// Mitsubishi GX Works2 project: A01_20260228_0   PLC: Q03UDV

TYPE arrange : STRUCT
  層 : ARRAY [1..5] OF STRING[12] := [5('')];
END_STRUCT END_TYPE

TYPE arrange_Bit : STRUCT
  層 : ARRAY [1..5] OF BOOL;
END_STRUCT END_TYPE

TYPE Master_R : STRUCT
  Stacker_Status : WORD;
  Aut_Process : INT;
  Error_Code : INT;
  Task_Status : WORD;
  現在Task_ID : DWORD;
  Task実行総数 : DINT;
  現在位置走行 : INT;
  現在位置リフト : INT;
  現在位置フォーク : INT;
  現在速度走行 : INT;
  現在速度リフト : INT;
  現在速度フォーク : INT;
  現在モード : INT;
  Heartbeat : INT;
  入庫要求1 : INT;
  入庫要求2 : INT;
  出庫要求1 : INT;
  出庫要求2 : INT;
  トルクX軸 : INT;
  トルクY軸 : INT;
  トルクZ軸 : INT;
  異常X軸 : INT;
  異常Y軸 : INT;
  異常Z軸 : INT;
  現在_列 : INT;
  現在_層 : INT;
  Status_Bit : INT;
  Warning_Code : INT;
END_STRUCT END_TYPE

TYPE Master_W : STRUCT
  Task_Type : WORD;
  Task_ID : DWORD;
  起点棚 : INT;
  起点列 : INT;
  起点層 : INT;
  終点棚 : INT;
  終点列 : INT;
  終点層 : INT;
  搬入ST_NO : INT;
  搬出ST_NO : INT;
  System_Heartbeat : INT;
  B01_搬入可 : INT;
  B02_搬入可 : INT;
  B01_搬出可 : INT;
  B02_搬出可 : INT;
  Mode : INT;
  REST_Cont : INT;
  一時停止_Cont : INT;
  Xj軸定位置 : INT;
  Y軸定位置 : INT;
  Z軸定位置 : INT;
  X軸定位列 : INT;
  Y軸定位層 : INT;
  Control_Bit : INT;
  緊急停止 : INT;
  Spare_16 : INT;
  Spare_17 : INT;
  Spare_18 : INT;
  Spare_19 : INT;
END_STRUCT END_TYPE

TYPE Single_Machine : STRUCT
  Query : BOOL;
  成功 : BOOL;
  棚場所 : INT;
  列場所 : INT;
  層場所 : INT;
  搬出PB : BOOL;
  RFID入力 : STRING[12];
  失敗 : BOOL;
  AGV行先 : INT;
  搬出許可条件 : BOOL;
  搬出口 : INT;
  搬出起点Status : INT;
  搬出終点Status : INT;
  搬入ST_パレットStatus : INT;
  搬出ST_パレットStatus : INT;
  搬出起点Status表示 : BOOL;
  終点搬入Status表示 : BOOL;
  搬入ST_Status表示 : BOOL;
  搬出ST_Status表示 : BOOL;
  空き保管場所検索 : BOOL;
  保管条件可 : BOOL;
  搬入PB : BOOL;
  Command_Status : INT;
END_STRUCT END_TYPE

TYPE Wcs_W : STRUCT
  Task_Type : WORD;
  Task_ID : DWORD;
  起点棚 : INT;
  起点列 : INT;
  起点層 : INT;
  終点棚 : INT;
  終点列 : INT;
  終点層 : INT;
  搬入ST_NO : INT;
  搬出ST_NO : INT;
  System_Heartbeat : INT;
  B01_搬入可 : INT;
  B02_搬入可 : INT;
  B01_搬出可 : INT;
  B02_搬出可 : INT;
  異常リセット : INT;
  Spare_7 : INT;
  Spare_8 : INT;
  Spare_9 : INT;
  Spare_10 : INT;
  B01_AGV進入可 : INT;
  B02_AGV進入可 : INT;
  B01_搬入RFID異常 : INT;
  B01_搬出RFID異常 : INT;
  B02_搬入RFID異常 : INT;
  B02_搬出RFID異常 : INT;
  Spare_17 : INT;
  Spare_18 : INT;
  Spare_19 : INT;
END_STRUCT END_TYPE

// global labels: Global1
VAR_GLOBAL
  Stacker_R : Master_R;
  Stacker_W : Master_W;
  Wcs_W : Wcs_W;
  Alone : Wcs_W;
  Mode AT D450 : INT;
  inventory_1 : ARRAY [1..14] OF arrange;
  inventory_2 : ARRAY [1..14] OF arrange;
  搬入RFID_Coding : STRING[12];
  inventory_Bit1 : ARRAY [1..14] OF arrange_Bit;
  inventory_Bit2 : ARRAY [1..14] OF arrange_Bit;
  在庫クリア AT M205 : BOOL;
  Single_Machine : Single_Machine;
  B01CV_OutID : DWORD;
  B02CV_OutID : DWORD;
  Stacker_Done : BOOL;
END_VAR

PROGRAM 01  // PLC 入力
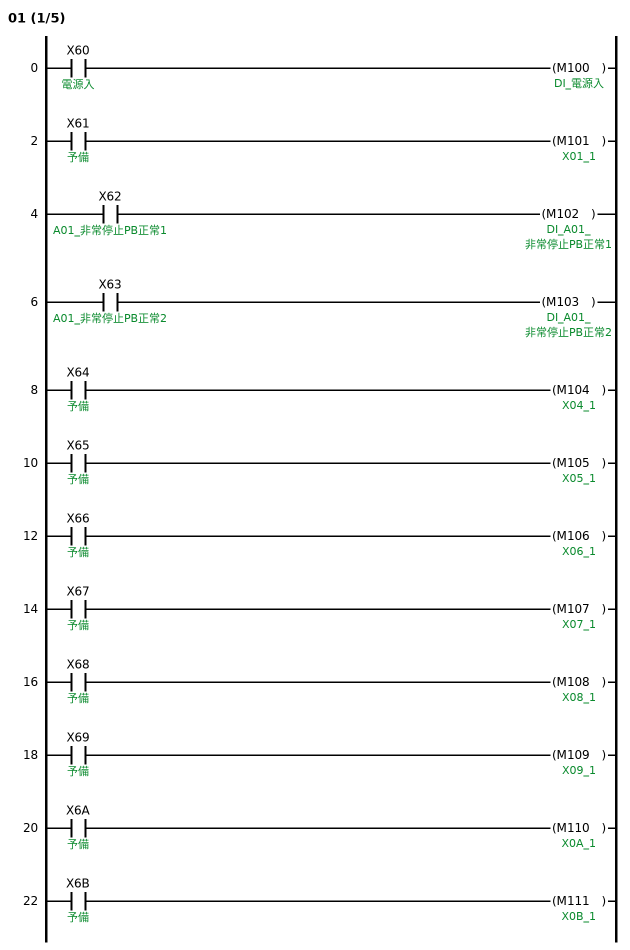
0     LD      X60  ; 電源入
      OUT     M100  ; DI_電源入
2     LD      X61  ; 予備
      OUT     M101  ; X01_1
4     LD      X62  ; A01_非常停止PB正常1
      OUT     M102  ; DI_A01_非常停止PB正常1
6     LD      X63  ; A01_非常停止PB正常2
      OUT     M103  ; DI_A01_非常停止PB正常2
8     LD      X64  ; 予備
      OUT     M104  ; X04_1
10    LD      X65  ; 予備
      OUT     M105  ; X05_1
12    LD      X66  ; 予備
      OUT     M106  ; X06_1
14    LD      X67  ; 予備
      OUT     M107  ; X07_1
16    LD      X68  ; 予備
      OUT     M108  ; X08_1
18    LD      X69  ; 予備
      OUT     M109  ; X09_1
20    LD      X6A  ; 予備
      OUT     M110  ; X0A_1
22    LD      X6B  ; 予備
      OUT     M111  ; X0B_1
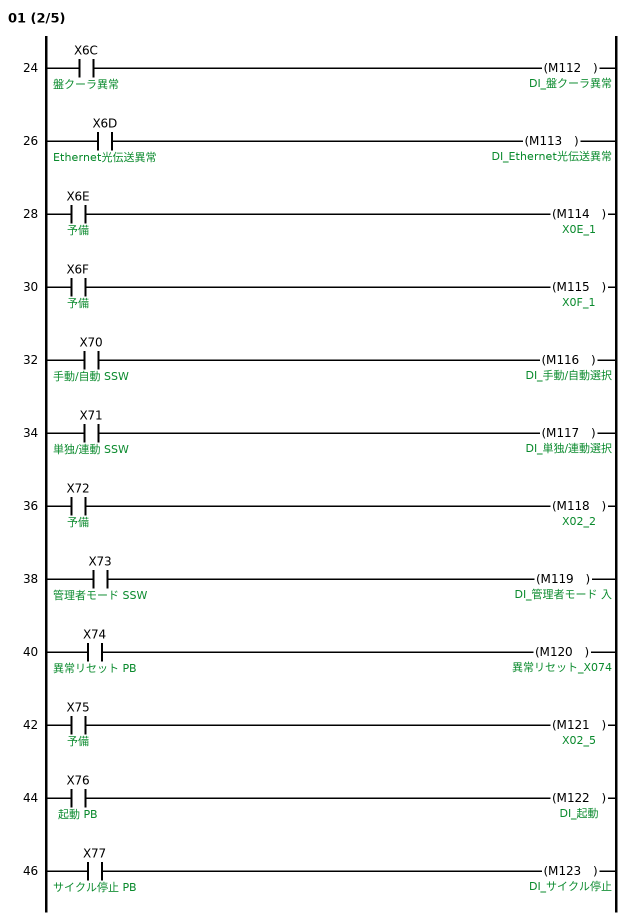
24    LD      X6C  ; 盤クーラ異常
      OUT     M112  ; DI_盤クーラ異常
26    LD      X6D  ; Ethernet光伝送異常
      OUT     M113  ; DI_Ethernet光伝送異常
28    LD      X6E  ; 予備
      OUT     M114  ; X0E_1
30    LD      X6F  ; 予備
      OUT     M115  ; X0F_1
32    LD      X70  ; 手動/自動 SSW
      OUT     M116  ; DI_手動/自動選択
34    LD      X71  ; 単独/連動 SSW
      OUT     M117  ; DI_単独/連動選択
36    LD      X72  ; 予備
      OUT     M118  ; X02_2
38    LD      X73  ; 管理者モード SSW
      OUT     M119  ; DI_管理者モード 入
40    LD      X74  ; 異常リセット PB
      OUT     M120  ; 異常リセット_X074
42    LD      X75  ; 予備
      OUT     M121  ; X02_5
44    LD      X76  ; 起動 PB
      OUT     M122  ; DI_起動
46    LD      X77  ; サイクル停止 PB
      OUT     M123  ; DI_サイクル停止
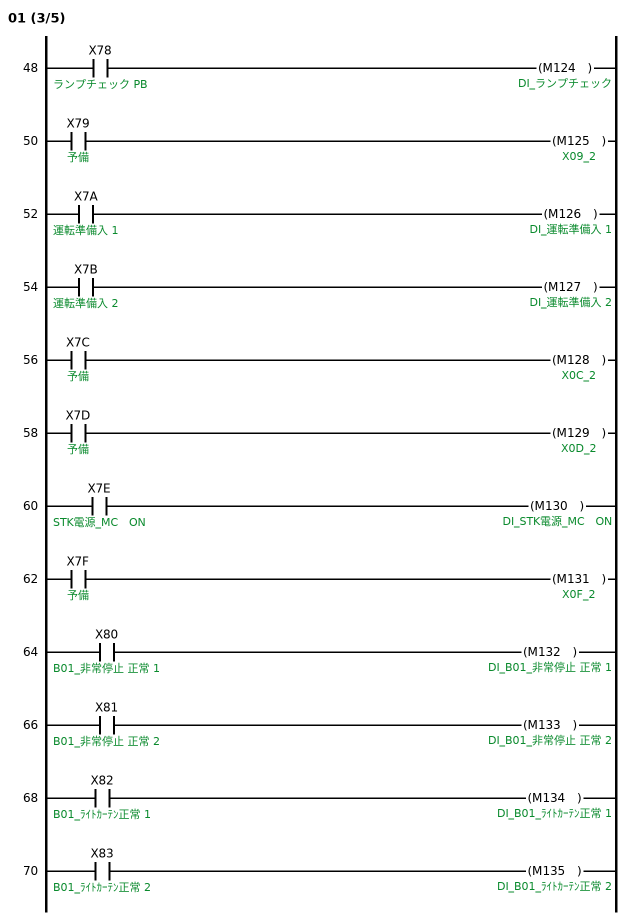
48    LD      X78  ; ランプチェック PB
      OUT     M124  ; DI_ランプチェック
50    LD      X79  ; 予備
      OUT     M125  ; X09_2
52    LD      X7A  ; 運転準備入 1
      OUT     M126  ; DI_運転準備入 1
54    LD      X7B  ; 運転準備入 2
      OUT     M127  ; DI_運転準備入 2
56    LD      X7C  ; 予備
      OUT     M128  ; X0C_2
58    LD      X7D  ; 予備
      OUT     M129  ; X0D_2
60    LD      X7E  ; STK電源_MC　ON
      OUT     M130  ; DI_STK電源_MC　ON
62    LD      X7F  ; 予備
      OUT     M131  ; X0F_2
64    LD      X80  ; B01_非常停止 正常 1
      OUT     M132  ; DI_B01_非常停止 正常 1
66    LD      X81  ; B01_非常停止 正常 2
      OUT     M133  ; DI_B01_非常停止 正常 2
68    LD      X82  ; B01_ﾗｲﾄｶｰﾃﾝ正常 1
      OUT     M134  ; DI_B01_ﾗｲﾄｶｰﾃﾝ正常 1
70    LD      X83  ; B01_ﾗｲﾄｶｰﾃﾝ正常 2
      OUT     M135  ; DI_B01_ﾗｲﾄｶｰﾃﾝ正常 2
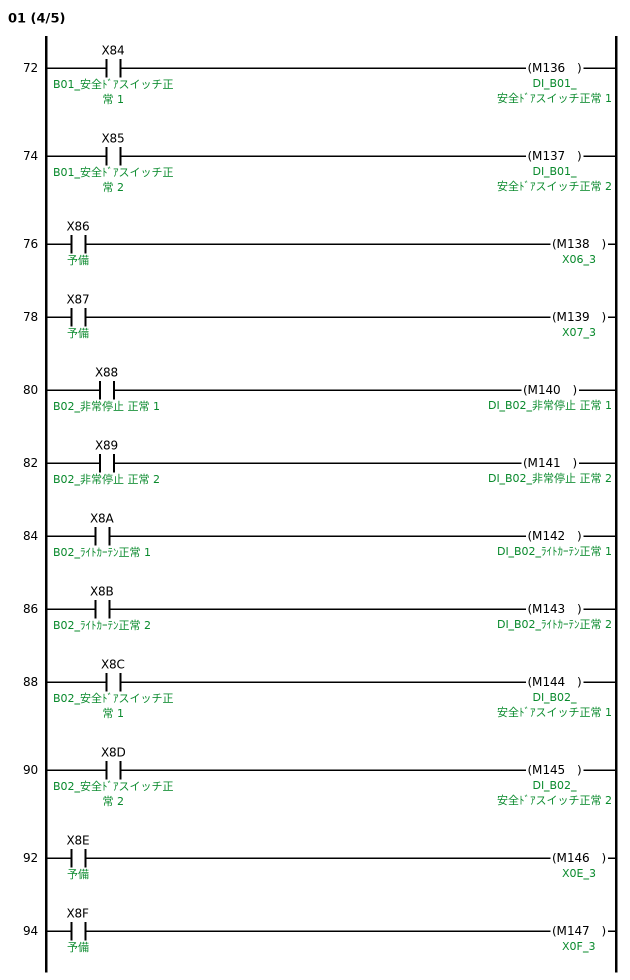
72    LD      X84  ; B01_安全ﾄﾞｱスイッチ正常 1
      OUT     M136  ; DI_B01_安全ﾄﾞｱスイッチ正常 1
74    LD      X85  ; B01_安全ﾄﾞｱスイッチ正常 2
      OUT     M137  ; DI_B01_安全ﾄﾞｱスイッチ正常 2
76    LD      X86  ; 予備
      OUT     M138  ; X06_3
78    LD      X87  ; 予備
      OUT     M139  ; X07_3
80    LD      X88  ; B02_非常停止 正常 1
      OUT     M140  ; DI_B02_非常停止 正常 1
82    LD      X89  ; B02_非常停止 正常 2
      OUT     M141  ; DI_B02_非常停止 正常 2
84    LD      X8A  ; B02_ﾗｲﾄｶｰﾃﾝ正常 1
      OUT     M142  ; DI_B02_ﾗｲﾄｶｰﾃﾝ正常 1
86    LD      X8B  ; B02_ﾗｲﾄｶｰﾃﾝ正常 2
      OUT     M143  ; DI_B02_ﾗｲﾄｶｰﾃﾝ正常 2
88    LD      X8C  ; B02_安全ﾄﾞｱスイッチ正常 1
      OUT     M144  ; DI_B02_安全ﾄﾞｱスイッチ正常 1
90    LD      X8D  ; B02_安全ﾄﾞｱスイッチ正常 2
      OUT     M145  ; DI_B02_安全ﾄﾞｱスイッチ正常 2
92    LD      X8E  ; 予備
      OUT     M146  ; X0E_3
94    LD      X8F  ; 予備
      OUT     M147  ; X0F_3
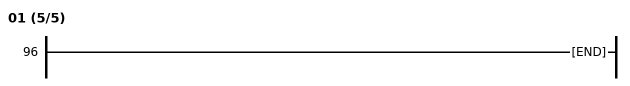
96    END
END_PROGRAM

PROGRAM 02  // スタッカー 入力
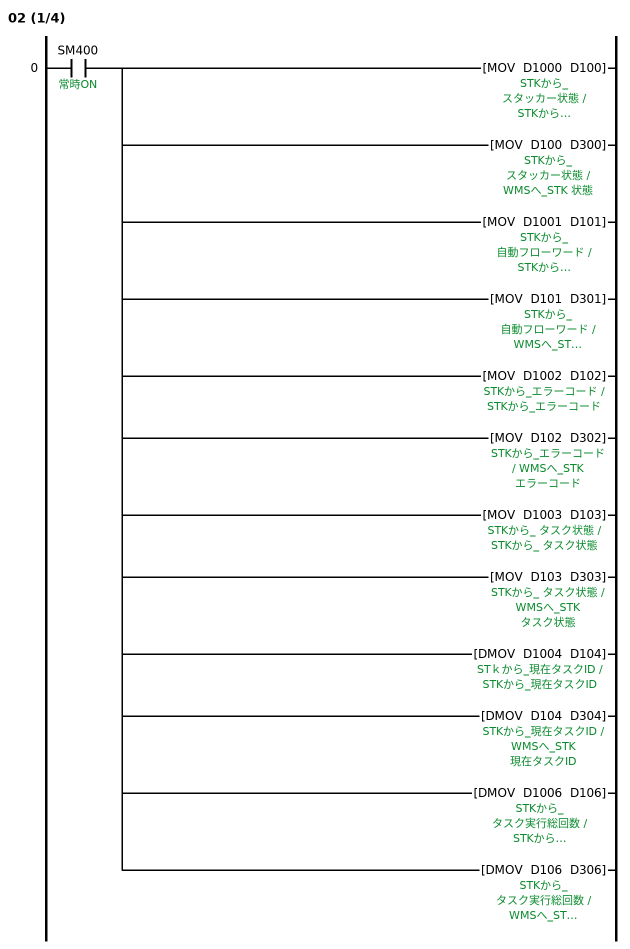
0     LD      SM400  ; 常時ON
      MOV     D1000 D100  ; STKから_スタッカー状態 / STKから_スタッカー状態
      MOV     D100 D300  ; WMSへ_STK 状態
      MOV     D1001 D101  ; STKから_自動フローワード / STKから_自動フローワード
      MOV     D101 D301  ; WMSへ_STK 自動フローワード
      MOV     D1002 D102  ; STKから_エラーコード / STKから_エラーコード
      MOV     D102 D302  ; WMSへ_STK エラーコード
      MOV     D1003 D103  ; STKから_ タスク状態 / STKから_ タスク状態
      MOV     D103 D303  ; WMSへ_STK タスク状態
      DMOV    D1004 D104  ; STｋから_現在タスクID / STKから_現在タスクID
      DMOV    D104 D304  ; WMSへ_STK 現在タスクID
      DMOV    D1006 D106  ; STKから_タスク実行総回数 / STKから_タスク実行総回数
      DMOV    D106 D306  ; WMSへ_STK タスク実行総回数
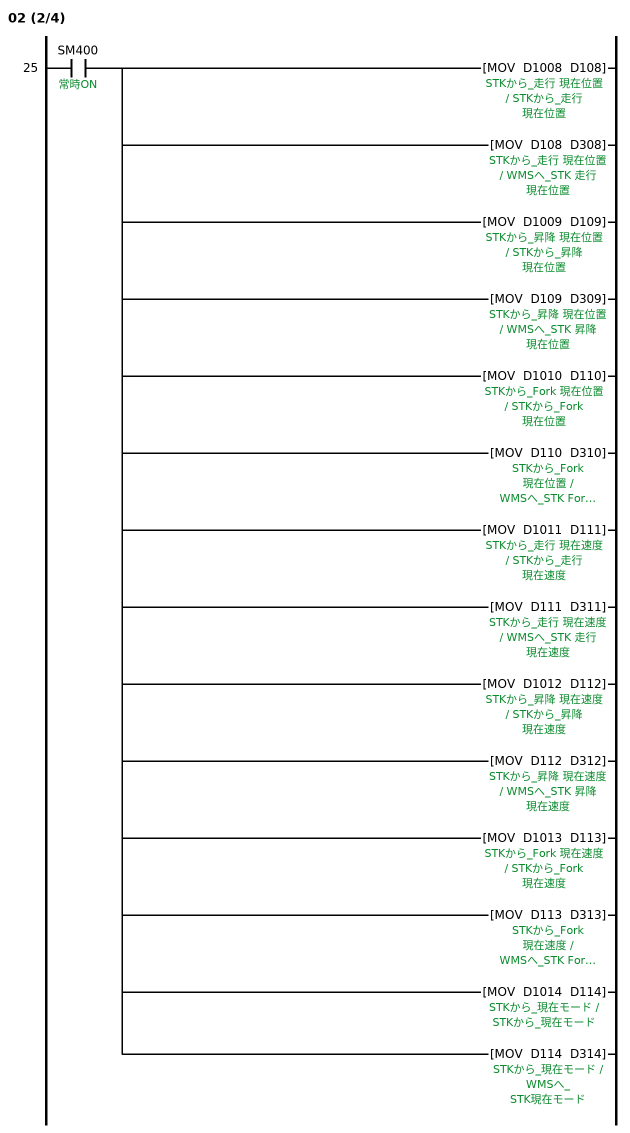
25    LD      SM400  ; 常時ON
      MOV     D1008 D108  ; STKから_走行 現在位置 / STKから_走行 現在位置
      MOV     D108 D308  ; WMSへ_STK 走行 現在位置
      MOV     D1009 D109  ; STKから_昇降 現在位置 / STKから_昇降 現在位置
      MOV     D109 D309  ; WMSへ_STK 昇降 現在位置
      MOV     D1010 D110  ; STKから_Fork 現在位置 / STKから_Fork 現在位置
      MOV     D110 D310  ; WMSへ_STK Fork 現在位置
      MOV     D1011 D111  ; STKから_走行 現在速度 / STKから_走行 現在速度
      MOV     D111 D311  ; WMSへ_STK 走行 現在速度
      MOV     D1012 D112  ; STKから_昇降 現在速度 / STKから_昇降 現在速度
      MOV     D112 D312  ; WMSへ_STK 昇降 現在速度
      MOV     D1013 D113  ; STKから_Fork 現在速度 / STKから_Fork 現在速度
      MOV     D113 D313  ; WMSへ_STK Fork 現在速度
      MOV     D1014 D114  ; STKから_現在モード / STKから_現在モード
      MOV     D114 D314  ; WMSへ_STK現在モード
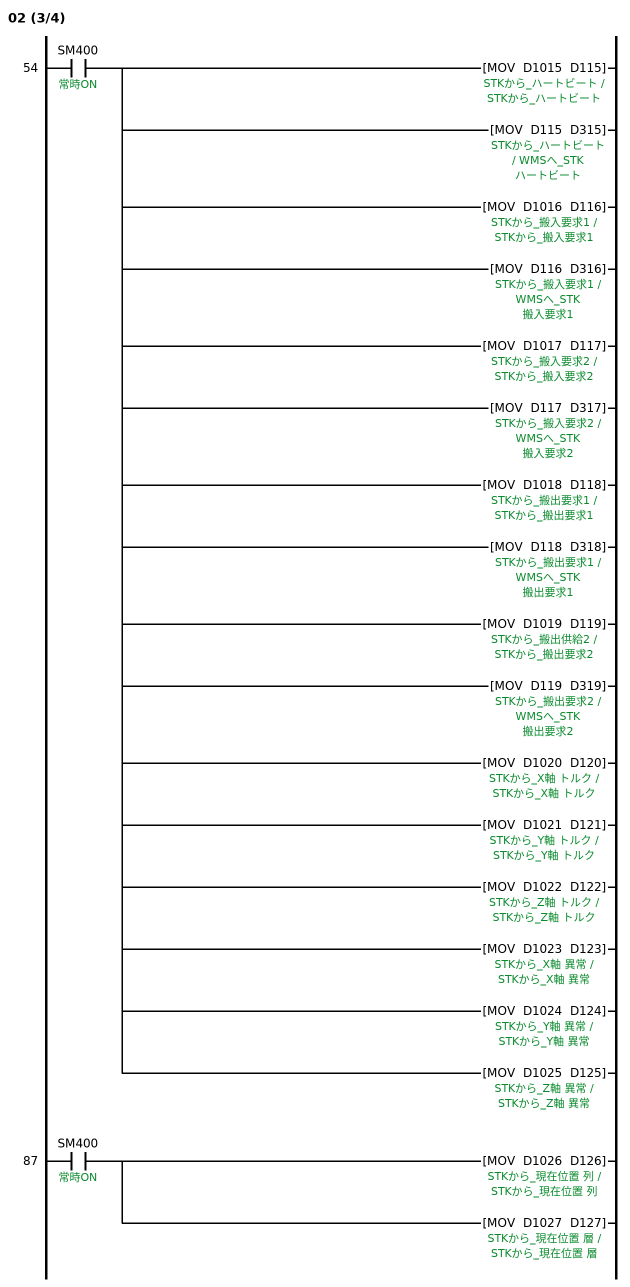
54    LD      SM400  ; 常時ON
      MOV     D1015 D115  ; STKから_ハートビート / STKから_ハートビート
      MOV     D115 D315  ; WMSへ_STK ハートビート
      MOV     D1016 D116  ; STKから_搬入要求1 / STKから_搬入要求1
      MOV     D116 D316  ; WMSへ_STK 搬入要求1
      MOV     D1017 D117  ; STKから_搬入要求2 / STKから_搬入要求2
      MOV     D117 D317  ; WMSへ_STK 搬入要求2
      MOV     D1018 D118  ; STKから_搬出要求1 / STKから_搬出要求1
      MOV     D118 D318  ; WMSへ_STK 搬出要求1
      MOV     D1019 D119  ; STKから_搬出供給2 / STKから_搬出要求2
      MOV     D119 D319  ; WMSへ_STK 搬出要求2
      MOV     D1020 D120  ; STKから_X軸 トルク / STKから_X軸 トルク
      MOV     D1021 D121  ; STKから_Y軸 トルク / STKから_Y軸 トルク
      MOV     D1022 D122  ; STKから_Z軸 トルク / STKから_Z軸 トルク
      MOV     D1023 D123  ; STKから_X軸 異常 / STKから_X軸 異常
      MOV     D1024 D124  ; STKから_Y軸 異常 / STKから_Y軸 異常
      MOV     D1025 D125  ; STKから_Z軸 異常 / STKから_Z軸 異常
87    LD      SM400  ; 常時ON
      MOV     D1026 D126  ; STKから_現在位置 列 / STKから_現在位置 列
      MOV     D1027 D127  ; STKから_現在位置 層 / STKから_現在位置 層
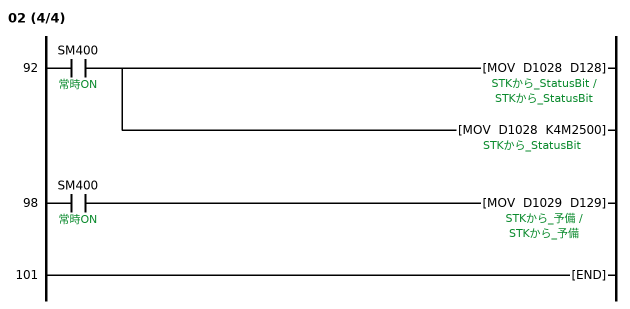
92    LD      SM400  ; 常時ON
      MOV     D1028 D128  ; STKから_StatusBit / STKから_StatusBit
      MOV     D1028 K4M2500  ; STKから_地面手動制御中
98    LD      SM400  ; 常時ON
      MOV     D1029 D129  ; STKから_予備 / STKから_予備
101   END
END_PROGRAM

PROGRAM 03  // WMS 入力
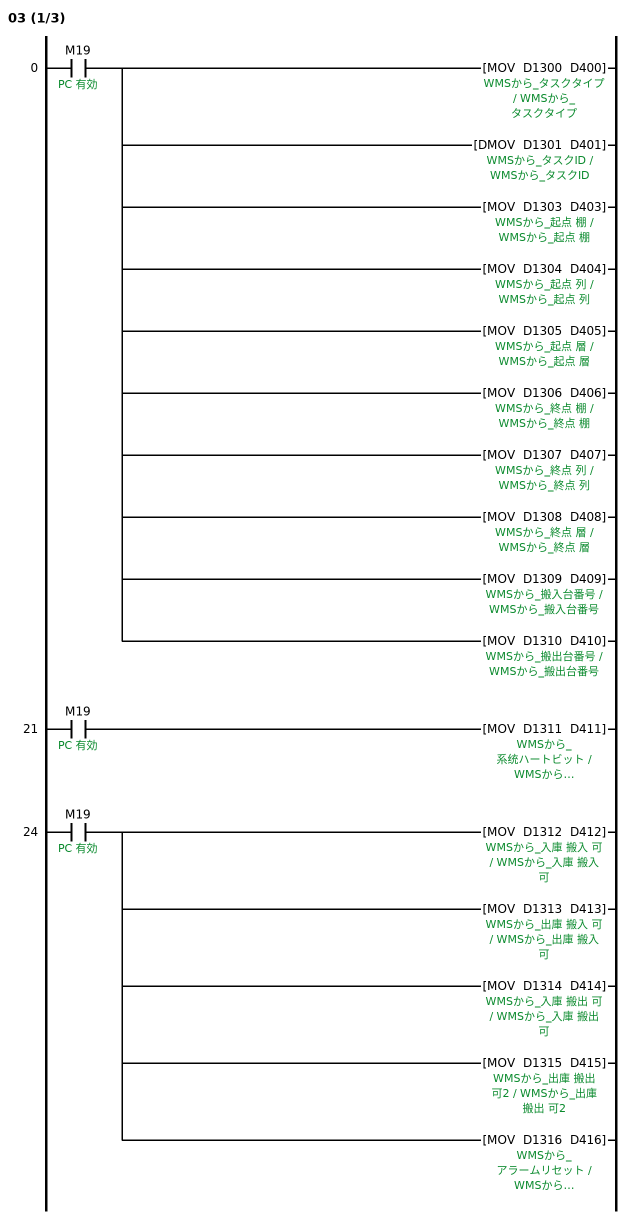
0     LD      M19  ; PC 有効
      MOV     D1300 D400  ; WMSから_タスクタイプ / WMSから_タスクタイプ
      DMOV    D1301 D401  ; WMSから_タスクID / WMSから_タスクID
      MOV     D1303 D403  ; WMSから_起点 棚 / WMSから_起点 棚
      MOV     D1304 D404  ; WMSから_起点 列 / WMSから_起点 列
      MOV     D1305 D405  ; WMSから_起点 層 / WMSから_起点 層
      MOV     D1306 D406  ; WMSから_終点 棚 / WMSから_終点 棚
      MOV     D1307 D407  ; WMSから_終点 列 / WMSから_終点 列
      MOV     D1308 D408  ; WMSから_終点 層 / WMSから_終点 層
      MOV     D1309 D409  ; WMSから_搬入台番号 / WMSから_搬入台番号
      MOV     D1310 D410  ; WMSから_搬出台番号 / WMSから_搬出台番号
21    LD      M19  ; PC 有効
      MOV     D1311 D411  ; WMSから_系统ハートビット / WMSから_系统ハートビット
24    LD      M19  ; PC 有効
      MOV     D1312 D412  ; WMSから_入庫 搬入 可 / WMSから_入庫 搬入 可
      MOV     D1313 D413  ; WMSから_出庫 搬入 可 / WMSから_出庫 搬入 可
      MOV     D1314 D414  ; WMSから_入庫 搬出 可 / WMSから_入庫 搬出 可
      MOV     D1315 D415  ; WMSから_出庫 搬出 可2 / WMSから_出庫 搬出 可2
      MOV     D1316 D416  ; WMSから_アラームリセット / WMSから_アラームリセット
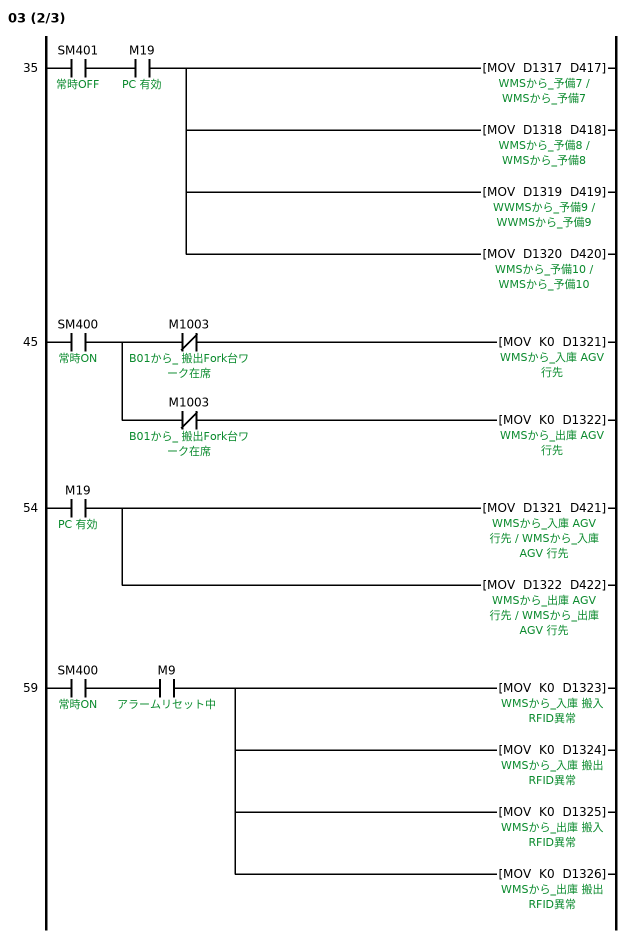
35    LD      SM401  ; 常時OFF
      AND     M19  ; PC 有効
      MOV     D1317 D417  ; WMSから_予備7 / WMSから_予備7
      MOV     D1318 D418  ; WMSから_予備8 / WMSから_予備8
      MOV     D1319 D419  ; WWMSから_予備9 / WWMSから_予備9
      MOV     D1320 D420  ; WMSから_予備10 / WMSから_予備10
45    LD      SM400  ; 常時ON
      MPS
      ANI     M1003  ; B01から_ 搬出Fork台ワーク在席
      MOV     K0 D1321  ; WMSから_入庫 AGV 行先
      MPP
      ANI     M1003  ; B01から_ 搬出Fork台ワーク在席
      MOV     K0 D1322  ; WMSから_出庫 AGV 行先
54    LD      M19  ; PC 有効
      MOV     D1321 D421  ; WMSから_入庫 AGV 行先
      MOV     D1322 D422  ; WMSから_出庫 AGV 行先
59    LD      SM400  ; 常時ON
      AND     M9  ; アラームリセット中
      MOV     K0 D1323  ; WMSから_入庫 搬入 RFID異常
      MOV     K0 D1324  ; WMSから_入庫 搬出 RFID異常
      MOV     K0 D1325  ; WMSから_出庫 搬入 RFID異常
      MOV     K0 D1326  ; WMSから_出庫 搬出 RFID異常
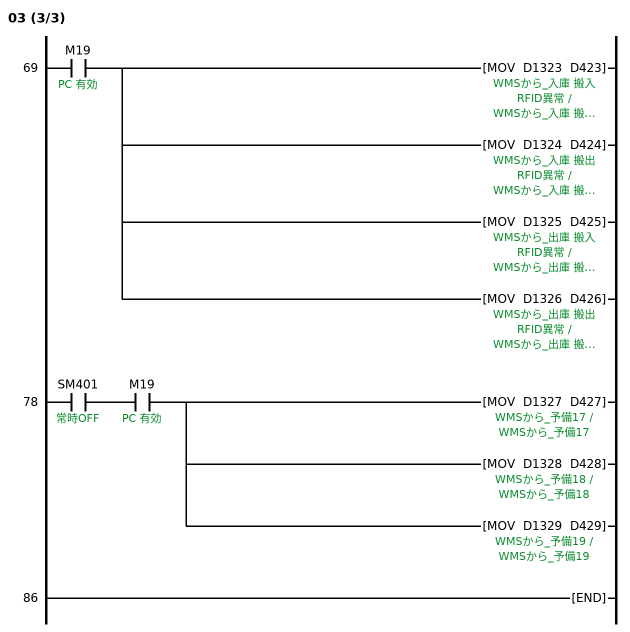
69    LD      M19  ; PC 有効
      MOV     D1323 D423  ; WMSから_入庫 搬入 RFID異常
      MOV     D1324 D424  ; WMSから_入庫 搬出 RFID異常
      MOV     D1325 D425  ; WMSから_出庫 搬入 RFID異常
      MOV     D1326 D426  ; WMSから_出庫 搬出 RFID異常
78    LD      SM401  ; 常時OFF
      AND     M19  ; PC 有効
      MOV     D1327 D427  ; WMSから_予備17 / WMSから_予備17
      MOV     D1328 D428  ; WMSから_予備18 / WMSから_予備18
      MOV     D1329 D429  ; WMSから_予備19 / WMSから_予備19
86    END
END_PROGRAM

PROGRAM 09  // 異常
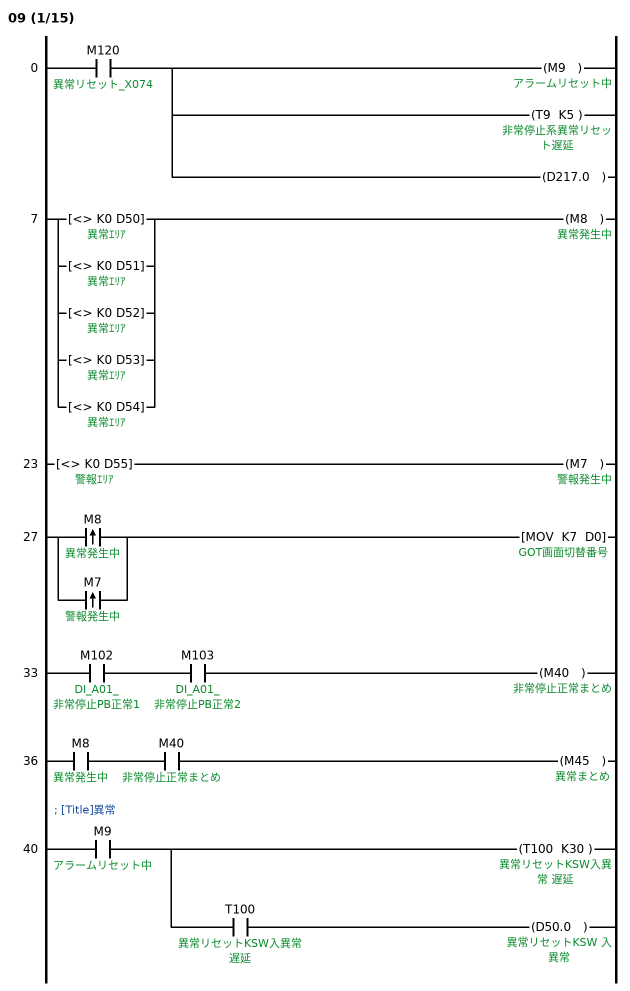
0     LD      M120  ; 異常リセット_X074
      OUT     M9  ; アラームリセット中
      OUT     T9 K5  ; 非常停止系異常リセット遅延
      OUT     D217.0
7     LD<>    K0 D50  ; 異常ｴﾘｱ
      OR<>    K0 D51  ; 異常ｴﾘｱ
      OR<>    K0 D52  ; 異常ｴﾘｱ
      OR<>    K0 D53  ; 異常ｴﾘｱ
      OR<>    K0 D54  ; 異常ｴﾘｱ
      OUT     M8  ; 異常発生中
23    LD<>    K0 D55  ; 警報ｴﾘｱ
      OUT     M7  ; 警報発生中
27    LDP     M8  ; 異常発生中
      ORP     M7  ; 警報発生中
      MOV     K7 D0  ; GOT画面切替番号
33    LD      M102  ; DI_A01_非常停止PB正常1
      AND     M103  ; DI_A01_非常停止PB正常2
      OUT     M40  ; 非常停止正常まとめ
36    LD      M8  ; 異常発生中
      AND     M40  ; 非常停止正常まとめ
      OUT     M45  ; 異常まとめ
; [Title]異常
40    LD      M9  ; アラームリセット中
      OUT     T100 K30  ; 異常リセットKSW入異常 遅延
      AND     T100  ; 異常リセットKSW入異常 遅延
      OUT     D50.0  ; 異常リセットKSW 入 異常
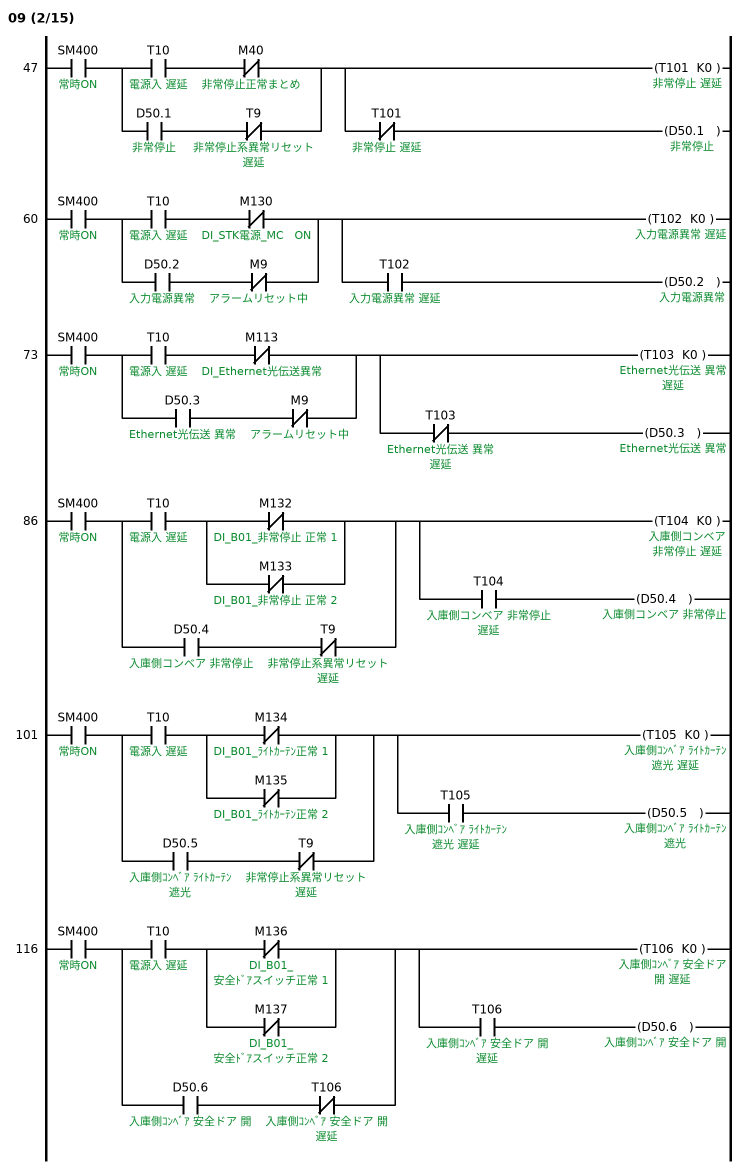
47    LD      SM400  ; 常時ON
      LD      T10  ; 電源入 遅延
      ANI     M40  ; 非常停止正常まとめ
      LD      D50.1  ; 非常停止
      ANI     T9  ; 非常停止系異常リセット遅延
      ORB
      ANB
      OUT     T101 K0  ; 非常停止 遅延
      ANI     T101  ; 非常停止 遅延
      OUT     D50.1  ; 非常停止
60    LD      SM400  ; 常時ON
      LD      T10  ; 電源入 遅延
      ANI     M130  ; DI_STK電源_MC　ON
      LD      D50.2  ; 入力電源異常
      ANI     M9  ; アラームリセット中
      ORB
      ANB
      OUT     T102 K0  ; 入力電源異常 遅延
      AND     T102  ; 入力電源異常 遅延
      OUT     D50.2  ; 入力電源異常
73    LD      SM400  ; 常時ON
      LD      T10  ; 電源入 遅延
      ANI     M113  ; DI_Ethernet光伝送異常
      LD      D50.3  ; Ethernet光伝送 異常
      ANI     M9  ; アラームリセット中
      ORB
      ANB
      OUT     T103 K0  ; Ethernet光伝送 異常 遅延
      ANI     T103  ; Ethernet光伝送 異常 遅延
      OUT     D50.3  ; Ethernet光伝送 異常
86    LD      SM400  ; 常時ON
      LD      T10  ; 電源入 遅延
      LDI     M132  ; DI_B01_非常停止 正常 1
      ORI     M133  ; DI_B01_非常停止 正常 2
      ANB
      LD      D50.4  ; 入庫側コンベア 非常停止
      ANI     T9  ; 非常停止系異常リセット遅延
      ORB
      ANB
      OUT     T104 K0  ; 入庫側コンベア 非常停止 遅延
      AND     T104  ; 入庫側コンベア 非常停止 遅延
      OUT     D50.4  ; 入庫側コンベア 非常停止
101   LD      SM400  ; 常時ON
      LD      T10  ; 電源入 遅延
      LDI     M134  ; DI_B01_ﾗｲﾄｶｰﾃﾝ正常 1
      ORI     M135  ; DI_B01_ﾗｲﾄｶｰﾃﾝ正常 2
      ANB
      LD      D50.5  ; 入庫側ｺﾝﾍﾞｱ ﾗｲﾄｶｰﾃﾝ 遮光
      ANI     T9  ; 非常停止系異常リセット遅延
      ORB
      ANB
      OUT     T105 K0  ; 入庫側ｺﾝﾍﾞｱ ﾗｲﾄｶｰﾃﾝ 遮光 遅延
      AND     T105  ; 入庫側ｺﾝﾍﾞｱ ﾗｲﾄｶｰﾃﾝ 遮光 遅延
      OUT     D50.5  ; 入庫側ｺﾝﾍﾞｱ ﾗｲﾄｶｰﾃﾝ 遮光
116   LD      SM400  ; 常時ON
      LD      T10  ; 電源入 遅延
      LDI     M136  ; DI_B01_安全ﾄﾞｱスイッチ正常 1
      ORI     M137  ; DI_B01_安全ﾄﾞｱスイッチ正常 2
      ANB
      LD      D50.6  ; 入庫側ｺﾝﾍﾞｱ 安全ドア 開
      ANI     T106  ; 入庫側ｺﾝﾍﾞｱ 安全ドア 開 遅延
      ORB
      ANB
      OUT     T106 K0  ; 入庫側ｺﾝﾍﾞｱ 安全ドア 開 遅延
      AND     T106  ; 入庫側ｺﾝﾍﾞｱ 安全ドア 開 遅延
      OUT     D50.6  ; 入庫側ｺﾝﾍﾞｱ 安全ドア 開
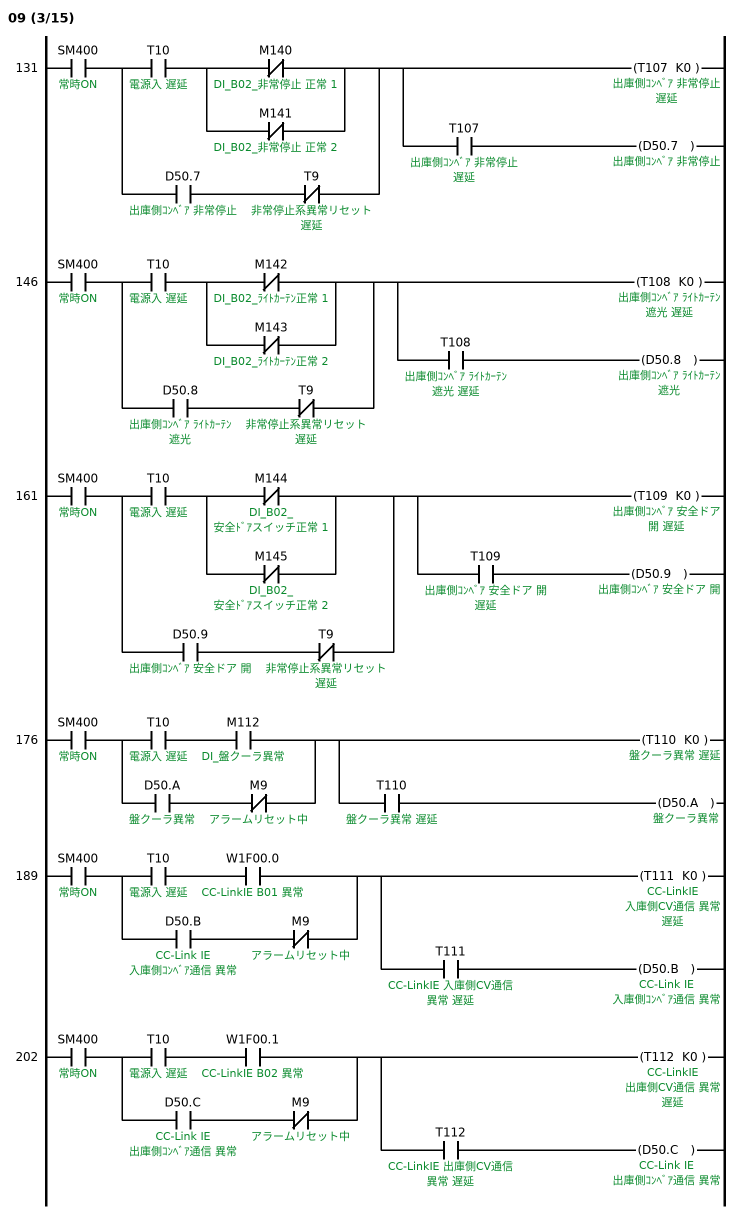
131   LD      SM400  ; 常時ON
      LD      T10  ; 電源入 遅延
      LDI     M140  ; DI_B02_非常停止 正常 1
      ORI     M141  ; DI_B02_非常停止 正常 2
      ANB
      LD      D50.7  ; 出庫側ｺﾝﾍﾞｱ 非常停止
      ANI     T9  ; 非常停止系異常リセット遅延
      ORB
      ANB
      OUT     T107 K0  ; 出庫側ｺﾝﾍﾞｱ 非常停止 遅延
      AND     T107  ; 出庫側ｺﾝﾍﾞｱ 非常停止 遅延
      OUT     D50.7  ; 出庫側ｺﾝﾍﾞｱ 非常停止
146   LD      SM400  ; 常時ON
      LD      T10  ; 電源入 遅延
      LDI     M142  ; DI_B02_ﾗｲﾄｶｰﾃﾝ正常 1
      ORI     M143  ; DI_B02_ﾗｲﾄｶｰﾃﾝ正常 2
      ANB
      LD      D50.8  ; 出庫側ｺﾝﾍﾞｱ ﾗｲﾄｶｰﾃﾝ 遮光
      ANI     T9  ; 非常停止系異常リセット遅延
      ORB
      ANB
      OUT     T108 K0  ; 出庫側ｺﾝﾍﾞｱ ﾗｲﾄｶｰﾃﾝ 遮光 遅延
      AND     T108  ; 出庫側ｺﾝﾍﾞｱ ﾗｲﾄｶｰﾃﾝ 遮光 遅延
      OUT     D50.8  ; 出庫側ｺﾝﾍﾞｱ ﾗｲﾄｶｰﾃﾝ 遮光
161   LD      SM400  ; 常時ON
      LD      T10  ; 電源入 遅延
      LDI     M144  ; DI_B02_安全ﾄﾞｱスイッチ正常 1
      ORI     M145  ; DI_B02_安全ﾄﾞｱスイッチ正常 2
      ANB
      LD      D50.9  ; 出庫側ｺﾝﾍﾞｱ 安全ドア 開
      ANI     T9  ; 非常停止系異常リセット遅延
      ORB
      ANB
      OUT     T109 K0  ; 出庫側ｺﾝﾍﾞｱ 安全ドア 開 遅延
      AND     T109  ; 出庫側ｺﾝﾍﾞｱ 安全ドア 開 遅延
      OUT     D50.9  ; 出庫側ｺﾝﾍﾞｱ 安全ドア 開
176   LD      SM400  ; 常時ON
      LD      T10  ; 電源入 遅延
      AND     M112  ; DI_盤クーラ異常
      LD      D50.A  ; 盤クーラ異常
      ANI     M9  ; アラームリセット中
      ORB
      ANB
      OUT     T110 K0  ; 盤クーラ異常 遅延
      AND     T110  ; 盤クーラ異常 遅延
      OUT     D50.A  ; 盤クーラ異常
189   LD      SM400  ; 常時ON
      LD      T10  ; 電源入 遅延
      AND     W1F00.0  ; CC-LinkIE B01 異常
      LD      D50.B  ; CC-Link IE 入庫側ｺﾝﾍﾞｱ通信 異常
      ANI     M9  ; アラームリセット中
      ORB
      ANB
      OUT     T111 K0  ; CC-LinkIE 入庫側CV通信 異常 遅延
      AND     T111  ; CC-LinkIE 入庫側CV通信 異常 遅延
      OUT     D50.B  ; CC-Link IE 入庫側ｺﾝﾍﾞｱ通信 異常
202   LD      SM400  ; 常時ON
      LD      T10  ; 電源入 遅延
      AND     W1F00.1  ; CC-LinkIE B02 異常
      LD      D50.C  ; CC-Link IE 出庫側ｺﾝﾍﾞｱ通信 異常
      ANI     M9  ; アラームリセット中
      ORB
      ANB
      OUT     T112 K0  ; CC-LinkIE 出庫側CV通信 異常 遅延
      AND     T112  ; CC-LinkIE 出庫側CV通信 異常 遅延
      OUT     D50.C  ; CC-Link IE 出庫側ｺﾝﾍﾞｱ通信 異常
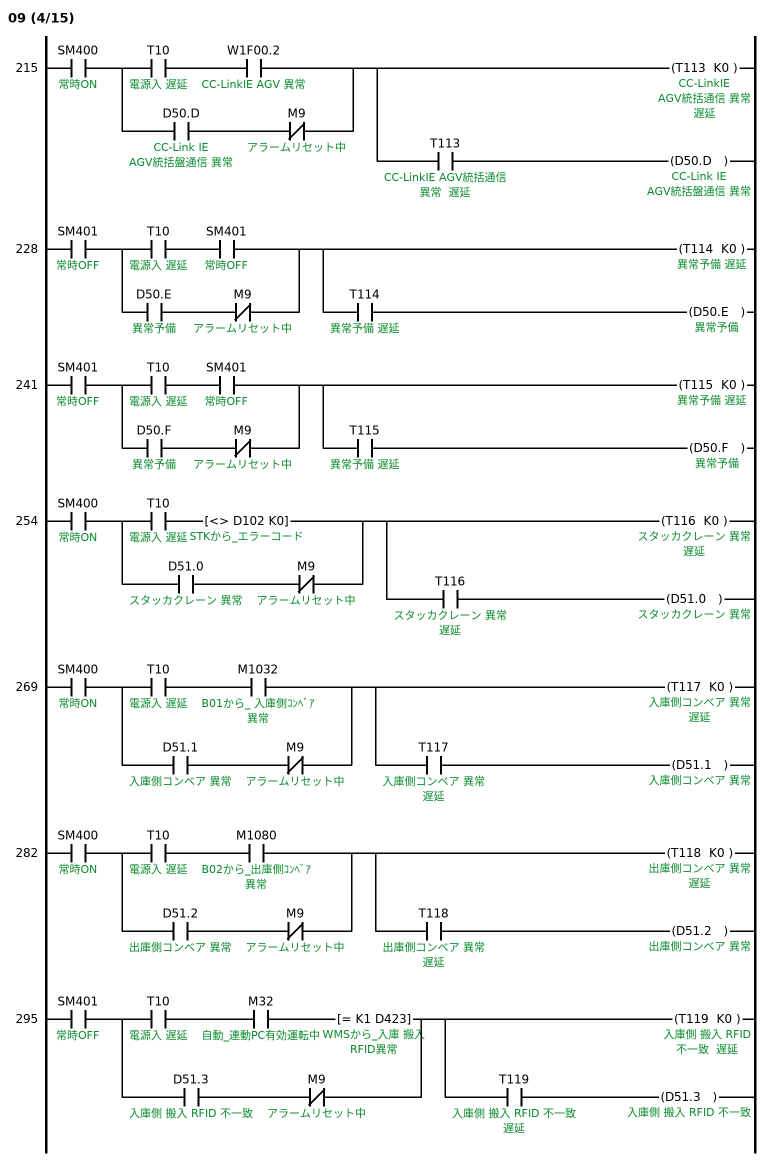
215   LD      SM400  ; 常時ON
      LD      T10  ; 電源入 遅延
      AND     W1F00.2  ; CC-LinkIE AGV 異常
      LD      D50.D  ; CC-Link IE AGV統括盤通信 異常
      ANI     M9  ; アラームリセット中
      ORB
      ANB
      OUT     T113 K0  ; CC-LinkIE AGV統括通信 異常  遅延
      AND     T113  ; CC-LinkIE AGV統括通信 異常  遅延
      OUT     D50.D  ; CC-Link IE AGV統括盤通信 異常
228   LD      SM401  ; 常時OFF
      LD      T10  ; 電源入 遅延
      AND     SM401  ; 常時OFF
      LD      D50.E  ; 異常予備
      ANI     M9  ; アラームリセット中
      ORB
      ANB
      OUT     T114 K0  ; 異常予備 遅延
      AND     T114  ; 異常予備 遅延
      OUT     D50.E  ; 異常予備
241   LD      SM401  ; 常時OFF
      LD      T10  ; 電源入 遅延
      AND     SM401  ; 常時OFF
      LD      D50.F  ; 異常予備
      ANI     M9  ; アラームリセット中
      ORB
      ANB
      OUT     T115 K0  ; 異常予備 遅延
      AND     T115  ; 異常予備 遅延
      OUT     D50.F  ; 異常予備
254   LD      SM400  ; 常時ON
      LD      T10  ; 電源入 遅延
      AND<>   D102 K0  ; STKから_エラーコード
      LD      D51.0  ; スタッカクレーン 異常
      ANI     M9  ; アラームリセット中
      ORB
      ANB
      OUT     T116 K0  ; スタッカクレーン 異常  遅延
      AND     T116  ; スタッカクレーン 異常  遅延
      OUT     D51.0  ; スタッカクレーン 異常
269   LD      SM400  ; 常時ON
      LD      T10  ; 電源入 遅延
      AND     M1032  ; B01から_ 入庫側ｺﾝﾍﾞｱ 異常
      LD      D51.1  ; 入庫側コンベア 異常
      ANI     M9  ; アラームリセット中
      ORB
      ANB
      OUT     T117 K0  ; 入庫側コンベア 異常  遅延
      AND     T117  ; 入庫側コンベア 異常  遅延
      OUT     D51.1  ; 入庫側コンベア 異常
282   LD      SM400  ; 常時ON
      LD      T10  ; 電源入 遅延
      AND     M1080  ; B02から_出庫側ｺﾝﾍﾞｱ 異常
      LD      D51.2  ; 出庫側コンベア 異常
      ANI     M9  ; アラームリセット中
      ORB
      ANB
      OUT     T118 K0  ; 出庫側コンベア 異常  遅延
      AND     T118  ; 出庫側コンベア 異常  遅延
      OUT     D51.2  ; 出庫側コンベア 異常
295   LD      SM401  ; 常時OFF
      LD      T10  ; 電源入 遅延
      AND     M32  ; 自動_連動PC有効運転中
      AND=    K1 D423  ; WMSから_入庫 搬入 RFID異常
      LD      D51.3  ; 入庫側 搬入 RFID 不一致
      ANI     M9  ; アラームリセット中
      ORB
      ANB
      OUT     T119 K0  ; 入庫側 搬入 RFID 不一致  遅延
      AND     T119  ; 入庫側 搬入 RFID 不一致  遅延
      OUT     D51.3  ; 入庫側 搬入 RFID 不一致
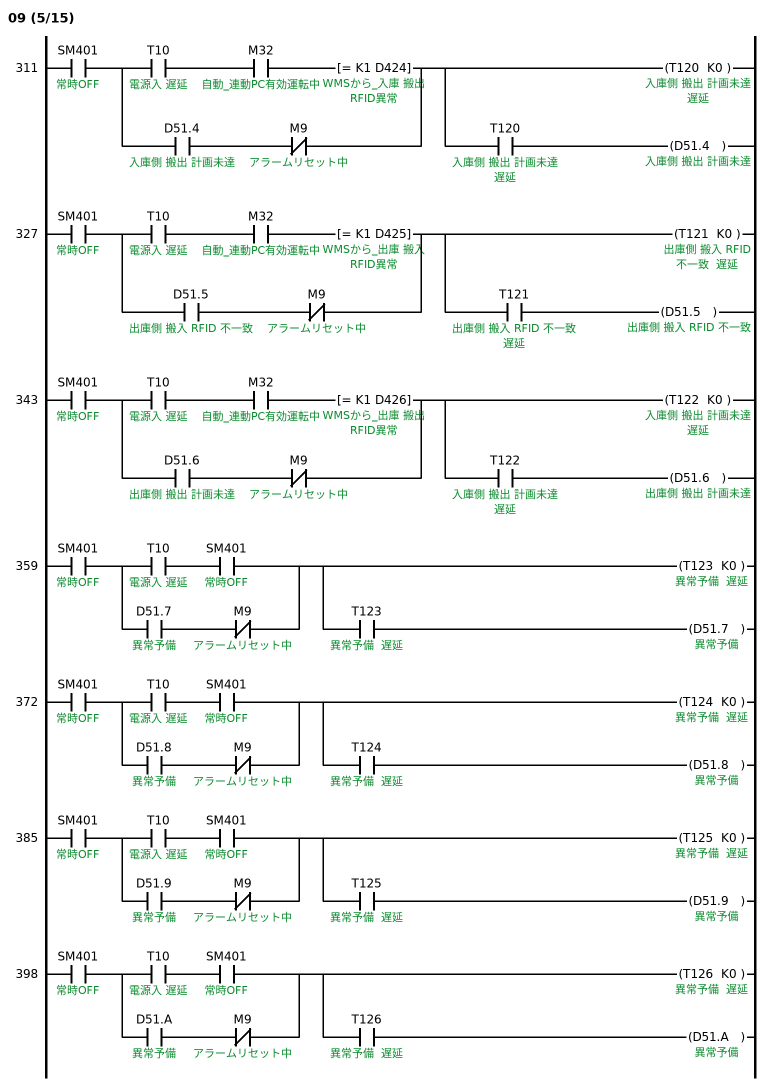
311   LD      SM401  ; 常時OFF
      LD      T10  ; 電源入 遅延
      AND     M32  ; 自動_連動PC有効運転中
      AND=    K1 D424  ; WMSから_入庫 搬出 RFID異常
      LD      D51.4  ; 入庫側 搬出 計画未達
      ANI     M9  ; アラームリセット中
      ORB
      ANB
      OUT     T120 K0  ; 入庫側 搬出 計画未達  遅延
      AND     T120  ; 入庫側 搬出 計画未達  遅延
      OUT     D51.4  ; 入庫側 搬出 計画未達
327   LD      SM401  ; 常時OFF
      LD      T10  ; 電源入 遅延
      AND     M32  ; 自動_連動PC有効運転中
      AND=    K1 D425  ; WMSから_出庫 搬入 RFID異常
      LD      D51.5  ; 出庫側 搬入 RFID 不一致
      ANI     M9  ; アラームリセット中
      ORB
      ANB
      OUT     T121 K0  ; 出庫側 搬入 RFID 不一致  遅延
      AND     T121  ; 出庫側 搬入 RFID 不一致  遅延
      OUT     D51.5  ; 出庫側 搬入 RFID 不一致
343   LD      SM401  ; 常時OFF
      LD      T10  ; 電源入 遅延
      AND     M32  ; 自動_連動PC有効運転中
      AND=    K1 D426  ; WMSから_出庫 搬出 RFID異常
      LD      D51.6  ; 出庫側 搬出 計画未達
      ANI     M9  ; アラームリセット中
      ORB
      ANB
      OUT     T122 K0  ; 入庫側 搬出 計画未達  遅延
      AND     T122  ; 入庫側 搬出 計画未達  遅延
      OUT     D51.6  ; 出庫側 搬出 計画未達
359   LD      SM401  ; 常時OFF
      LD      T10  ; 電源入 遅延
      AND     SM401  ; 常時OFF
      LD      D51.7  ; 異常予備
      ANI     M9  ; アラームリセット中
      ORB
      ANB
      OUT     T123 K0  ; 異常予備  遅延
      AND     T123  ; 異常予備  遅延
      OUT     D51.7  ; 異常予備
372   LD      SM401  ; 常時OFF
      LD      T10  ; 電源入 遅延
      AND     SM401  ; 常時OFF
      LD      D51.8  ; 異常予備
      ANI     M9  ; アラームリセット中
      ORB
      ANB
      OUT     T124 K0  ; 異常予備  遅延
      AND     T124  ; 異常予備  遅延
      OUT     D51.8  ; 異常予備
385   LD      SM401  ; 常時OFF
      LD      T10  ; 電源入 遅延
      AND     SM401  ; 常時OFF
      LD      D51.9  ; 異常予備
      ANI     M9  ; アラームリセット中
      ORB
      ANB
      OUT     T125 K0  ; 異常予備  遅延
      AND     T125  ; 異常予備  遅延
      OUT     D51.9  ; 異常予備
398   LD      SM401  ; 常時OFF
      LD      T10  ; 電源入 遅延
      AND     SM401  ; 常時OFF
      LD      D51.A  ; 異常予備
      ANI     M9  ; アラームリセット中
      ORB
      ANB
      OUT     T126 K0  ; 異常予備  遅延
      AND     T126  ; 異常予備  遅延
      OUT     D51.A  ; 異常予備
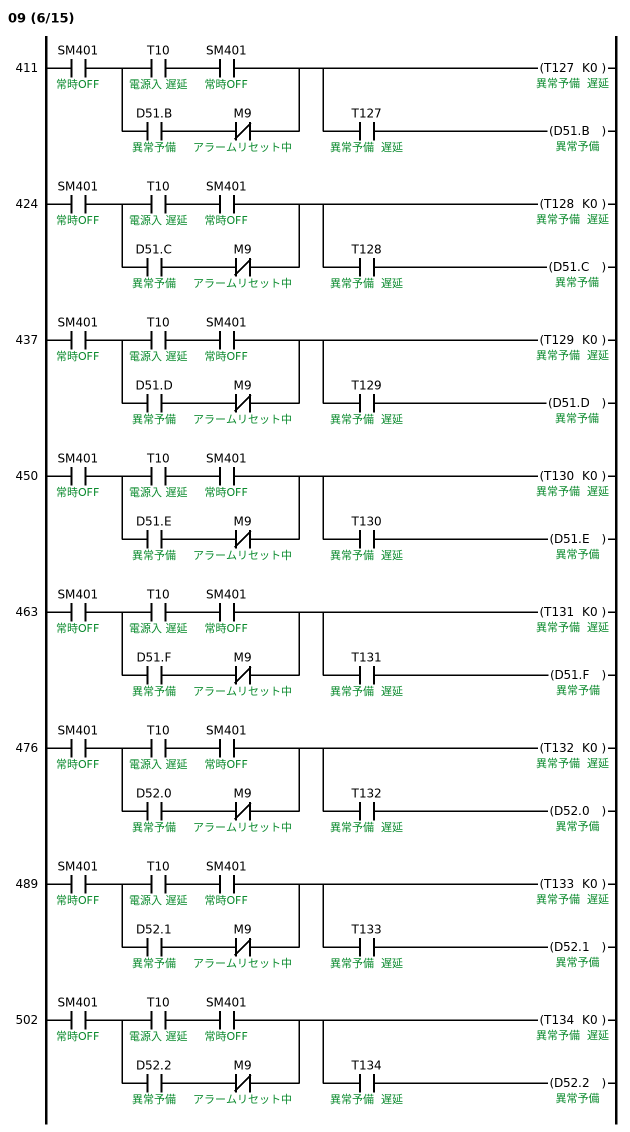
411   LD      SM401  ; 常時OFF
      LD      T10  ; 電源入 遅延
      AND     SM401  ; 常時OFF
      LD      D51.B  ; 異常予備
      ANI     M9  ; アラームリセット中
      ORB
      ANB
      OUT     T127 K0  ; 異常予備  遅延
      AND     T127  ; 異常予備  遅延
      OUT     D51.B  ; 異常予備
424   LD      SM401  ; 常時OFF
      LD      T10  ; 電源入 遅延
      AND     SM401  ; 常時OFF
      LD      D51.C  ; 異常予備
      ANI     M9  ; アラームリセット中
      ORB
      ANB
      OUT     T128 K0  ; 異常予備  遅延
      AND     T128  ; 異常予備  遅延
      OUT     D51.C  ; 異常予備
437   LD      SM401  ; 常時OFF
      LD      T10  ; 電源入 遅延
      AND     SM401  ; 常時OFF
      LD      D51.D  ; 異常予備
      ANI     M9  ; アラームリセット中
      ORB
      ANB
      OUT     T129 K0  ; 異常予備  遅延
      AND     T129  ; 異常予備  遅延
      OUT     D51.D  ; 異常予備
450   LD      SM401  ; 常時OFF
      LD      T10  ; 電源入 遅延
      AND     SM401  ; 常時OFF
      LD      D51.E  ; 異常予備
      ANI     M9  ; アラームリセット中
      ORB
      ANB
      OUT     T130 K0  ; 異常予備  遅延
      AND     T130  ; 異常予備  遅延
      OUT     D51.E  ; 異常予備
463   LD      SM401  ; 常時OFF
      LD      T10  ; 電源入 遅延
      AND     SM401  ; 常時OFF
      LD      D51.F  ; 異常予備
      ANI     M9  ; アラームリセット中
      ORB
      ANB
      OUT     T131 K0  ; 異常予備  遅延
      AND     T131  ; 異常予備  遅延
      OUT     D51.F  ; 異常予備
476   LD      SM401  ; 常時OFF
      LD      T10  ; 電源入 遅延
      AND     SM401  ; 常時OFF
      LD      D52.0  ; 異常予備
      ANI     M9  ; アラームリセット中
      ORB
      ANB
      OUT     T132 K0  ; 異常予備  遅延
      AND     T132  ; 異常予備  遅延
      OUT     D52.0  ; 異常予備
489   LD      SM401  ; 常時OFF
      LD      T10  ; 電源入 遅延
      AND     SM401  ; 常時OFF
      LD      D52.1  ; 異常予備
      ANI     M9  ; アラームリセット中
      ORB
      ANB
      OUT     T133 K0  ; 異常予備  遅延
      AND     T133  ; 異常予備  遅延
      OUT     D52.1  ; 異常予備
502   LD      SM401  ; 常時OFF
      LD      T10  ; 電源入 遅延
      AND     SM401  ; 常時OFF
      LD      D52.2  ; 異常予備
      ANI     M9  ; アラームリセット中
      ORB
      ANB
      OUT     T134 K0  ; 異常予備  遅延
      AND     T134  ; 異常予備  遅延
      OUT     D52.2  ; 異常予備
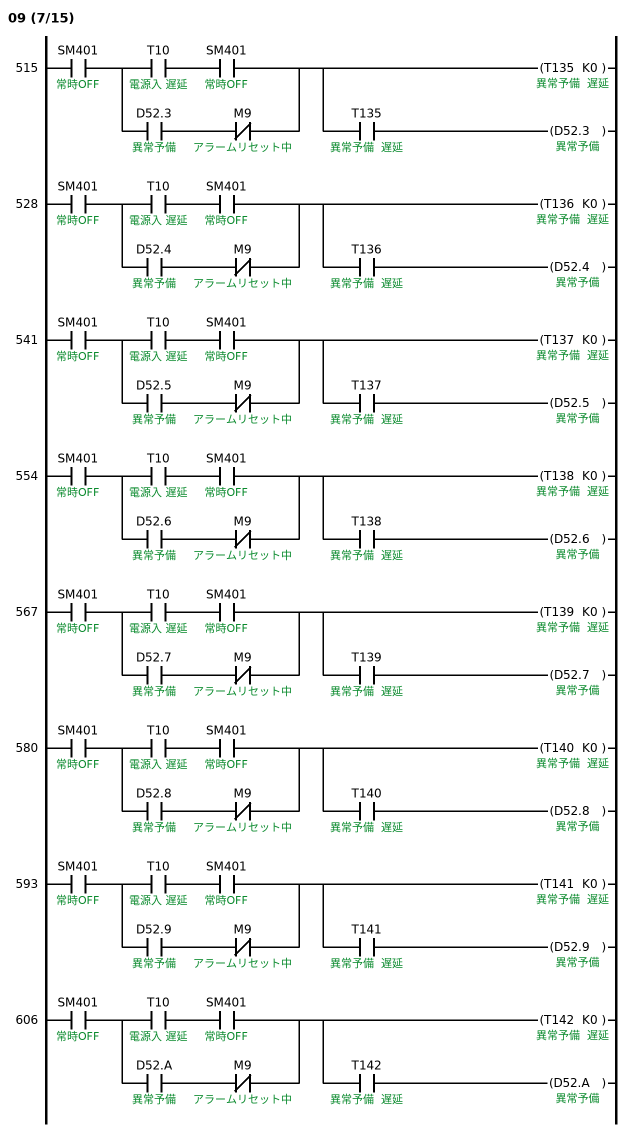
515   LD      SM401  ; 常時OFF
      LD      T10  ; 電源入 遅延
      AND     SM401  ; 常時OFF
      LD      D52.3  ; 異常予備
      ANI     M9  ; アラームリセット中
      ORB
      ANB
      OUT     T135 K0  ; 異常予備  遅延
      AND     T135  ; 異常予備  遅延
      OUT     D52.3  ; 異常予備
528   LD      SM401  ; 常時OFF
      LD      T10  ; 電源入 遅延
      AND     SM401  ; 常時OFF
      LD      D52.4  ; 異常予備
      ANI     M9  ; アラームリセット中
      ORB
      ANB
      OUT     T136 K0  ; 異常予備  遅延
      AND     T136  ; 異常予備  遅延
      OUT     D52.4  ; 異常予備
541   LD      SM401  ; 常時OFF
      LD      T10  ; 電源入 遅延
      AND     SM401  ; 常時OFF
      LD      D52.5  ; 異常予備
      ANI     M9  ; アラームリセット中
      ORB
      ANB
      OUT     T137 K0  ; 異常予備  遅延
      AND     T137  ; 異常予備  遅延
      OUT     D52.5  ; 異常予備
554   LD      SM401  ; 常時OFF
      LD      T10  ; 電源入 遅延
      AND     SM401  ; 常時OFF
      LD      D52.6  ; 異常予備
      ANI     M9  ; アラームリセット中
      ORB
      ANB
      OUT     T138 K0  ; 異常予備  遅延
      AND     T138  ; 異常予備  遅延
      OUT     D52.6  ; 異常予備
567   LD      SM401  ; 常時OFF
      LD      T10  ; 電源入 遅延
      AND     SM401  ; 常時OFF
      LD      D52.7  ; 異常予備
      ANI     M9  ; アラームリセット中
      ORB
      ANB
      OUT     T139 K0  ; 異常予備  遅延
      AND     T139  ; 異常予備  遅延
      OUT     D52.7  ; 異常予備
580   LD      SM401  ; 常時OFF
      LD      T10  ; 電源入 遅延
      AND     SM401  ; 常時OFF
      LD      D52.8  ; 異常予備
      ANI     M9  ; アラームリセット中
      ORB
      ANB
      OUT     T140 K0  ; 異常予備  遅延
      AND     T140  ; 異常予備  遅延
      OUT     D52.8  ; 異常予備
593   LD      SM401  ; 常時OFF
      LD      T10  ; 電源入 遅延
      AND     SM401  ; 常時OFF
      LD      D52.9  ; 異常予備
      ANI     M9  ; アラームリセット中
      ORB
      ANB
      OUT     T141 K0  ; 異常予備  遅延
      AND     T141  ; 異常予備  遅延
      OUT     D52.9  ; 異常予備
606   LD      SM401  ; 常時OFF
      LD      T10  ; 電源入 遅延
      AND     SM401  ; 常時OFF
      LD      D52.A  ; 異常予備
      ANI     M9  ; アラームリセット中
      ORB
      ANB
      OUT     T142 K0  ; 異常予備  遅延
      AND     T142  ; 異常予備  遅延
      OUT     D52.A  ; 異常予備
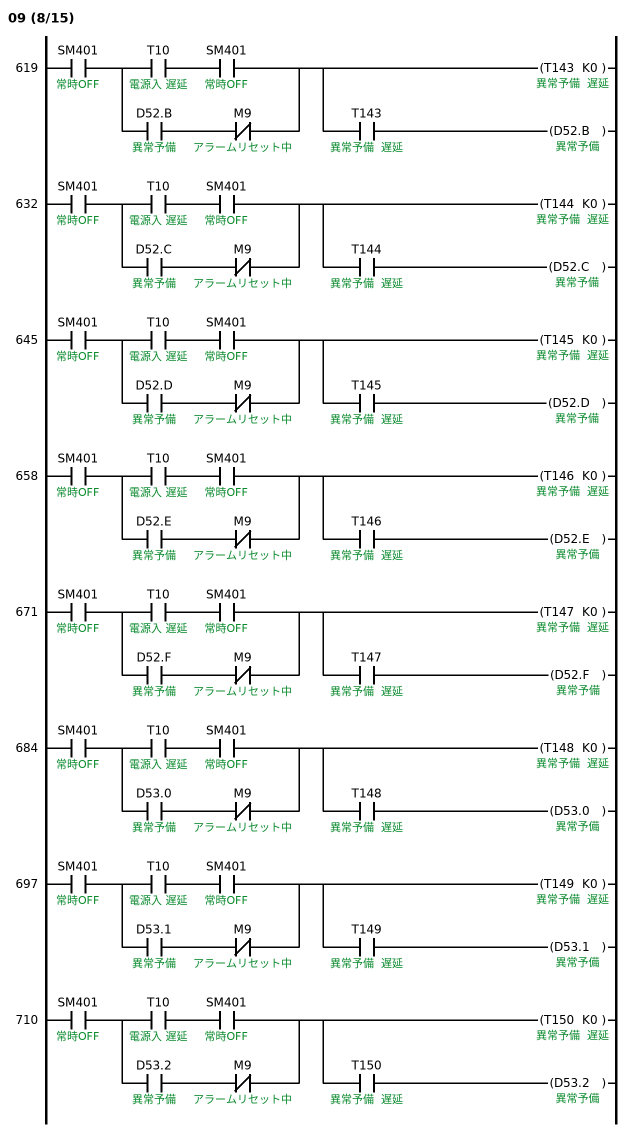
619   LD      SM401  ; 常時OFF
      LD      T10  ; 電源入 遅延
      AND     SM401  ; 常時OFF
      LD      D52.B  ; 異常予備
      ANI     M9  ; アラームリセット中
      ORB
      ANB
      OUT     T143 K0  ; 異常予備  遅延
      AND     T143  ; 異常予備  遅延
      OUT     D52.B  ; 異常予備
632   LD      SM401  ; 常時OFF
      LD      T10  ; 電源入 遅延
      AND     SM401  ; 常時OFF
      LD      D52.C  ; 異常予備
      ANI     M9  ; アラームリセット中
      ORB
      ANB
      OUT     T144 K0  ; 異常予備  遅延
      AND     T144  ; 異常予備  遅延
      OUT     D52.C  ; 異常予備
645   LD      SM401  ; 常時OFF
      LD      T10  ; 電源入 遅延
      AND     SM401  ; 常時OFF
      LD      D52.D  ; 異常予備
      ANI     M9  ; アラームリセット中
      ORB
      ANB
      OUT     T145 K0  ; 異常予備  遅延
      AND     T145  ; 異常予備  遅延
      OUT     D52.D  ; 異常予備
658   LD      SM401  ; 常時OFF
      LD      T10  ; 電源入 遅延
      AND     SM401  ; 常時OFF
      LD      D52.E  ; 異常予備
      ANI     M9  ; アラームリセット中
      ORB
      ANB
      OUT     T146 K0  ; 異常予備  遅延
      AND     T146  ; 異常予備  遅延
      OUT     D52.E  ; 異常予備
671   LD      SM401  ; 常時OFF
      LD      T10  ; 電源入 遅延
      AND     SM401  ; 常時OFF
      LD      D52.F  ; 異常予備
      ANI     M9  ; アラームリセット中
      ORB
      ANB
      OUT     T147 K0  ; 異常予備  遅延
      AND     T147  ; 異常予備  遅延
      OUT     D52.F  ; 異常予備
684   LD      SM401  ; 常時OFF
      LD      T10  ; 電源入 遅延
      AND     SM401  ; 常時OFF
      LD      D53.0  ; 異常予備
      ANI     M9  ; アラームリセット中
      ORB
      ANB
      OUT     T148 K0  ; 異常予備  遅延
      AND     T148  ; 異常予備  遅延
      OUT     D53.0  ; 異常予備
697   LD      SM401  ; 常時OFF
      LD      T10  ; 電源入 遅延
      AND     SM401  ; 常時OFF
      LD      D53.1  ; 異常予備
      ANI     M9  ; アラームリセット中
      ORB
      ANB
      OUT     T149 K0  ; 異常予備  遅延
      AND     T149  ; 異常予備  遅延
      OUT     D53.1  ; 異常予備
710   LD      SM401  ; 常時OFF
      LD      T10  ; 電源入 遅延
      AND     SM401  ; 常時OFF
      LD      D53.2  ; 異常予備
      ANI     M9  ; アラームリセット中
      ORB
      ANB
      OUT     T150 K0  ; 異常予備  遅延
      AND     T150  ; 異常予備  遅延
      OUT     D53.2  ; 異常予備
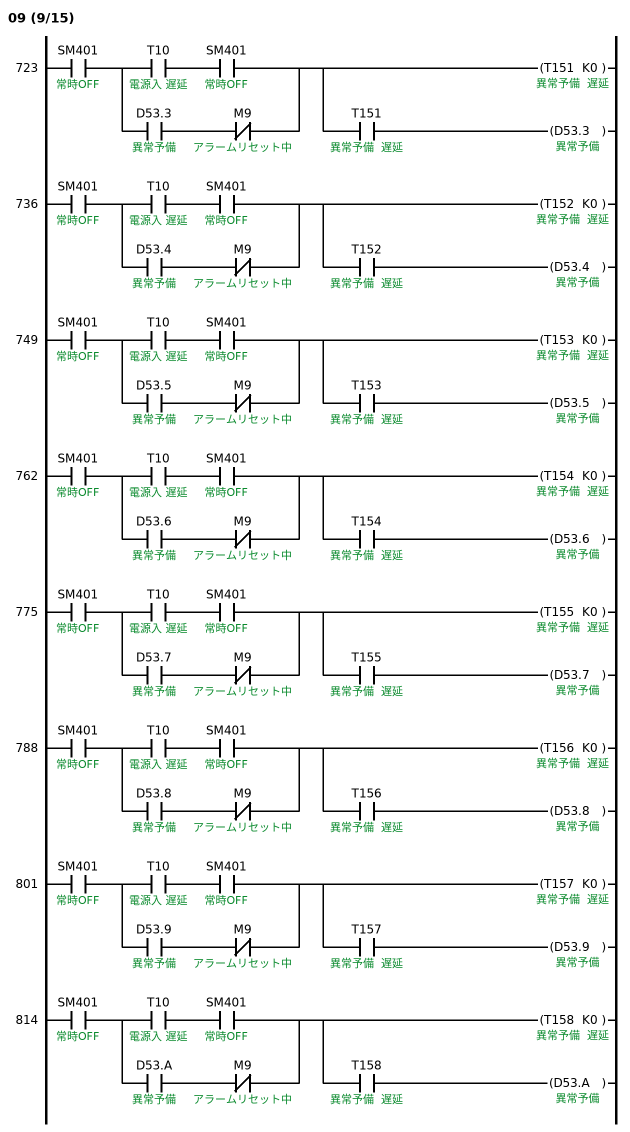
723   LD      SM401  ; 常時OFF
      LD      T10  ; 電源入 遅延
      AND     SM401  ; 常時OFF
      LD      D53.3  ; 異常予備
      ANI     M9  ; アラームリセット中
      ORB
      ANB
      OUT     T151 K0  ; 異常予備  遅延
      AND     T151  ; 異常予備  遅延
      OUT     D53.3  ; 異常予備
736   LD      SM401  ; 常時OFF
      LD      T10  ; 電源入 遅延
      AND     SM401  ; 常時OFF
      LD      D53.4  ; 異常予備
      ANI     M9  ; アラームリセット中
      ORB
      ANB
      OUT     T152 K0  ; 異常予備  遅延
      AND     T152  ; 異常予備  遅延
      OUT     D53.4  ; 異常予備
749   LD      SM401  ; 常時OFF
      LD      T10  ; 電源入 遅延
      AND     SM401  ; 常時OFF
      LD      D53.5  ; 異常予備
      ANI     M9  ; アラームリセット中
      ORB
      ANB
      OUT     T153 K0  ; 異常予備  遅延
      AND     T153  ; 異常予備  遅延
      OUT     D53.5  ; 異常予備
762   LD      SM401  ; 常時OFF
      LD      T10  ; 電源入 遅延
      AND     SM401  ; 常時OFF
      LD      D53.6  ; 異常予備
      ANI     M9  ; アラームリセット中
      ORB
      ANB
      OUT     T154 K0  ; 異常予備  遅延
      AND     T154  ; 異常予備  遅延
      OUT     D53.6  ; 異常予備
775   LD      SM401  ; 常時OFF
      LD      T10  ; 電源入 遅延
      AND     SM401  ; 常時OFF
      LD      D53.7  ; 異常予備
      ANI     M9  ; アラームリセット中
      ORB
      ANB
      OUT     T155 K0  ; 異常予備  遅延
      AND     T155  ; 異常予備  遅延
      OUT     D53.7  ; 異常予備
788   LD      SM401  ; 常時OFF
      LD      T10  ; 電源入 遅延
      AND     SM401  ; 常時OFF
      LD      D53.8  ; 異常予備
      ANI     M9  ; アラームリセット中
      ORB
      ANB
      OUT     T156 K0  ; 異常予備  遅延
      AND     T156  ; 異常予備  遅延
      OUT     D53.8  ; 異常予備
801   LD      SM401  ; 常時OFF
      LD      T10  ; 電源入 遅延
      AND     SM401  ; 常時OFF
      LD      D53.9  ; 異常予備
      ANI     M9  ; アラームリセット中
      ORB
      ANB
      OUT     T157 K0  ; 異常予備  遅延
      AND     T157  ; 異常予備  遅延
      OUT     D53.9  ; 異常予備
814   LD      SM401  ; 常時OFF
      LD      T10  ; 電源入 遅延
      AND     SM401  ; 常時OFF
      LD      D53.A  ; 異常予備
      ANI     M9  ; アラームリセット中
      ORB
      ANB
      OUT     T158 K0  ; 異常予備  遅延
      AND     T158  ; 異常予備  遅延
      OUT     D53.A  ; 異常予備
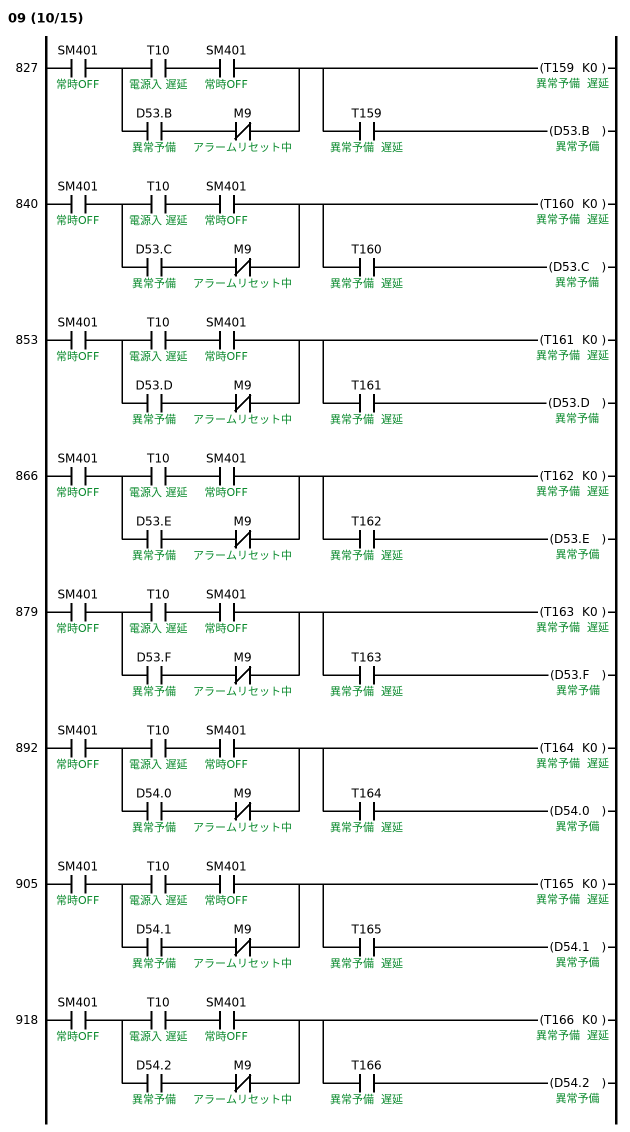
827   LD      SM401  ; 常時OFF
      LD      T10  ; 電源入 遅延
      AND     SM401  ; 常時OFF
      LD      D53.B  ; 異常予備
      ANI     M9  ; アラームリセット中
      ORB
      ANB
      OUT     T159 K0  ; 異常予備  遅延
      AND     T159  ; 異常予備  遅延
      OUT     D53.B  ; 異常予備
840   LD      SM401  ; 常時OFF
      LD      T10  ; 電源入 遅延
      AND     SM401  ; 常時OFF
      LD      D53.C  ; 異常予備
      ANI     M9  ; アラームリセット中
      ORB
      ANB
      OUT     T160 K0  ; 異常予備  遅延
      AND     T160  ; 異常予備  遅延
      OUT     D53.C  ; 異常予備
853   LD      SM401  ; 常時OFF
      LD      T10  ; 電源入 遅延
      AND     SM401  ; 常時OFF
      LD      D53.D  ; 異常予備
      ANI     M9  ; アラームリセット中
      ORB
      ANB
      OUT     T161 K0  ; 異常予備  遅延
      AND     T161  ; 異常予備  遅延
      OUT     D53.D  ; 異常予備
866   LD      SM401  ; 常時OFF
      LD      T10  ; 電源入 遅延
      AND     SM401  ; 常時OFF
      LD      D53.E  ; 異常予備
      ANI     M9  ; アラームリセット中
      ORB
      ANB
      OUT     T162 K0  ; 異常予備  遅延
      AND     T162  ; 異常予備  遅延
      OUT     D53.E  ; 異常予備
879   LD      SM401  ; 常時OFF
      LD      T10  ; 電源入 遅延
      AND     SM401  ; 常時OFF
      LD      D53.F  ; 異常予備
      ANI     M9  ; アラームリセット中
      ORB
      ANB
      OUT     T163 K0  ; 異常予備  遅延
      AND     T163  ; 異常予備  遅延
      OUT     D53.F  ; 異常予備
892   LD      SM401  ; 常時OFF
      LD      T10  ; 電源入 遅延
      AND     SM401  ; 常時OFF
      LD      D54.0  ; 異常予備
      ANI     M9  ; アラームリセット中
      ORB
      ANB
      OUT     T164 K0  ; 異常予備  遅延
      AND     T164  ; 異常予備  遅延
      OUT     D54.0  ; 異常予備
905   LD      SM401  ; 常時OFF
      LD      T10  ; 電源入 遅延
      AND     SM401  ; 常時OFF
      LD      D54.1  ; 異常予備
      ANI     M9  ; アラームリセット中
      ORB
      ANB
      OUT     T165 K0  ; 異常予備  遅延
      AND     T165  ; 異常予備  遅延
      OUT     D54.1  ; 異常予備
918   LD      SM401  ; 常時OFF
      LD      T10  ; 電源入 遅延
      AND     SM401  ; 常時OFF
      LD      D54.2  ; 異常予備
      ANI     M9  ; アラームリセット中
      ORB
      ANB
      OUT     T166 K0  ; 異常予備  遅延
      AND     T166  ; 異常予備  遅延
      OUT     D54.2  ; 異常予備
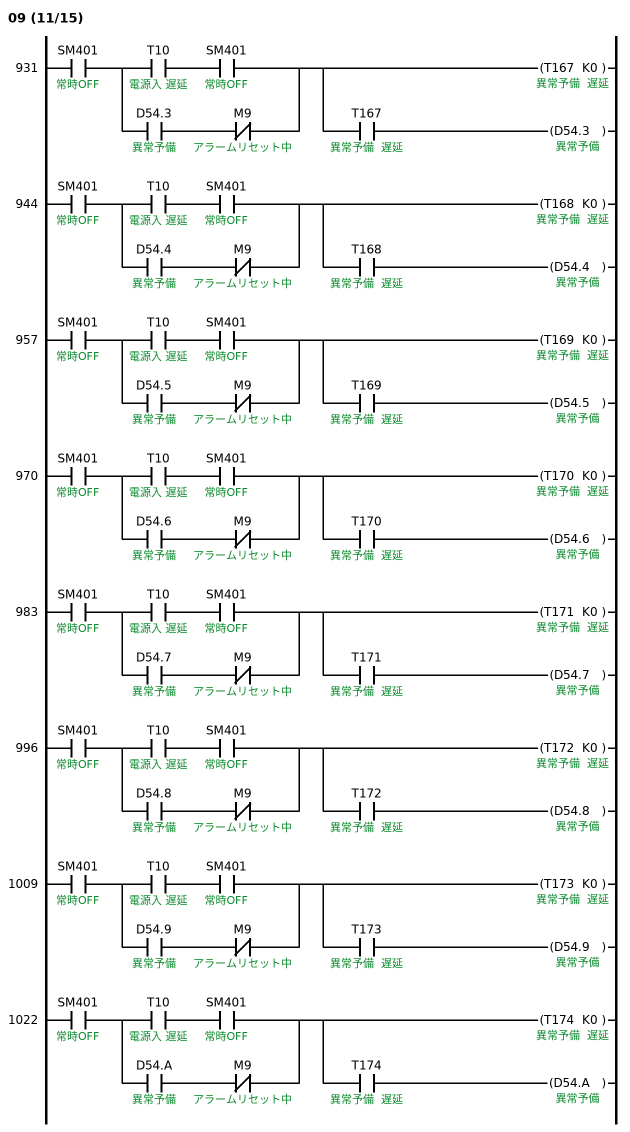
931   LD      SM401  ; 常時OFF
      LD      T10  ; 電源入 遅延
      AND     SM401  ; 常時OFF
      LD      D54.3  ; 異常予備
      ANI     M9  ; アラームリセット中
      ORB
      ANB
      OUT     T167 K0  ; 異常予備  遅延
      AND     T167  ; 異常予備  遅延
      OUT     D54.3  ; 異常予備
944   LD      SM401  ; 常時OFF
      LD      T10  ; 電源入 遅延
      AND     SM401  ; 常時OFF
      LD      D54.4  ; 異常予備
      ANI     M9  ; アラームリセット中
      ORB
      ANB
      OUT     T168 K0  ; 異常予備  遅延
      AND     T168  ; 異常予備  遅延
      OUT     D54.4  ; 異常予備
957   LD      SM401  ; 常時OFF
      LD      T10  ; 電源入 遅延
      AND     SM401  ; 常時OFF
      LD      D54.5  ; 異常予備
      ANI     M9  ; アラームリセット中
      ORB
      ANB
      OUT     T169 K0  ; 異常予備  遅延
      AND     T169  ; 異常予備  遅延
      OUT     D54.5  ; 異常予備
970   LD      SM401  ; 常時OFF
      LD      T10  ; 電源入 遅延
      AND     SM401  ; 常時OFF
      LD      D54.6  ; 異常予備
      ANI     M9  ; アラームリセット中
      ORB
      ANB
      OUT     T170 K0  ; 異常予備  遅延
      AND     T170  ; 異常予備  遅延
      OUT     D54.6  ; 異常予備
983   LD      SM401  ; 常時OFF
      LD      T10  ; 電源入 遅延
      AND     SM401  ; 常時OFF
      LD      D54.7  ; 異常予備
      ANI     M9  ; アラームリセット中
      ORB
      ANB
      OUT     T171 K0  ; 異常予備  遅延
      AND     T171  ; 異常予備  遅延
      OUT     D54.7  ; 異常予備
996   LD      SM401  ; 常時OFF
      LD      T10  ; 電源入 遅延
      AND     SM401  ; 常時OFF
      LD      D54.8  ; 異常予備
      ANI     M9  ; アラームリセット中
      ORB
      ANB
      OUT     T172 K0  ; 異常予備  遅延
      AND     T172  ; 異常予備  遅延
      OUT     D54.8  ; 異常予備
1009  LD      SM401  ; 常時OFF
      LD      T10  ; 電源入 遅延
      AND     SM401  ; 常時OFF
      LD      D54.9  ; 異常予備
      ANI     M9  ; アラームリセット中
      ORB
      ANB
      OUT     T173 K0  ; 異常予備  遅延
      AND     T173  ; 異常予備  遅延
      OUT     D54.9  ; 異常予備
1022  LD      SM401  ; 常時OFF
      LD      T10  ; 電源入 遅延
      AND     SM401  ; 常時OFF
      LD      D54.A  ; 異常予備
      ANI     M9  ; アラームリセット中
      ORB
      ANB
      OUT     T174 K0  ; 異常予備  遅延
      AND     T174  ; 異常予備  遅延
      OUT     D54.A  ; 異常予備
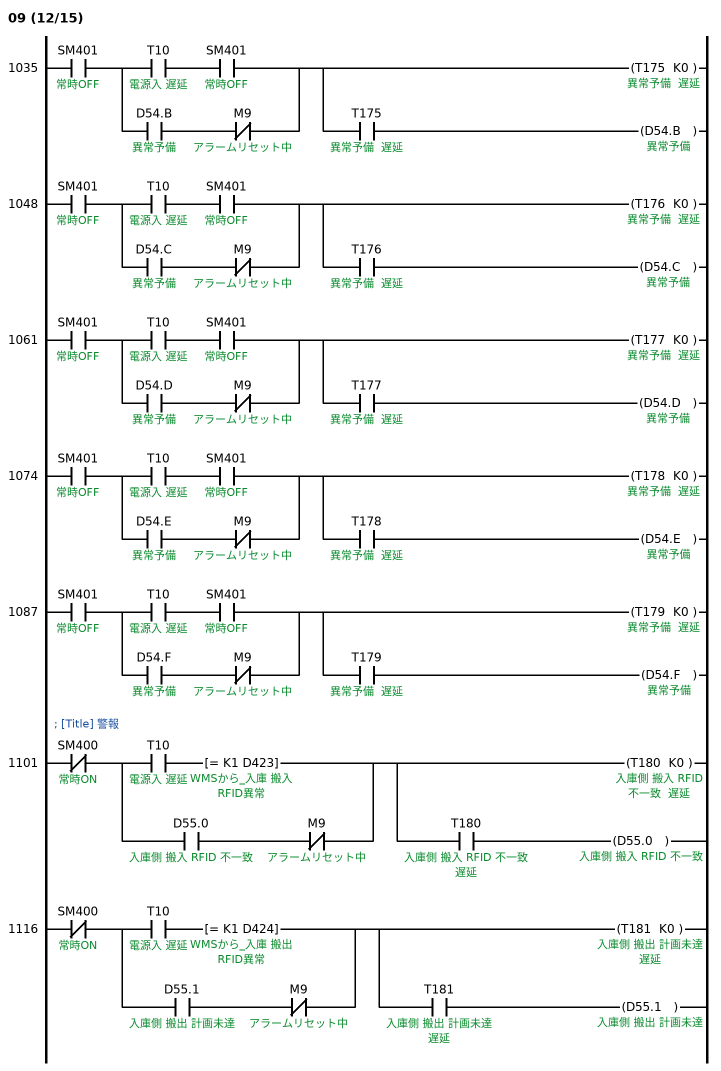
1035  LD      SM401  ; 常時OFF
      LD      T10  ; 電源入 遅延
      AND     SM401  ; 常時OFF
      LD      D54.B  ; 異常予備
      ANI     M9  ; アラームリセット中
      ORB
      ANB
      OUT     T175 K0  ; 異常予備  遅延
      AND     T175  ; 異常予備  遅延
      OUT     D54.B  ; 異常予備
1048  LD      SM401  ; 常時OFF
      LD      T10  ; 電源入 遅延
      AND     SM401  ; 常時OFF
      LD      D54.C  ; 異常予備
      ANI     M9  ; アラームリセット中
      ORB
      ANB
      OUT     T176 K0  ; 異常予備  遅延
      AND     T176  ; 異常予備  遅延
      OUT     D54.C  ; 異常予備
1061  LD      SM401  ; 常時OFF
      LD      T10  ; 電源入 遅延
      AND     SM401  ; 常時OFF
      LD      D54.D  ; 異常予備
      ANI     M9  ; アラームリセット中
      ORB
      ANB
      OUT     T177 K0  ; 異常予備  遅延
      AND     T177  ; 異常予備  遅延
      OUT     D54.D  ; 異常予備
1074  LD      SM401  ; 常時OFF
      LD      T10  ; 電源入 遅延
      AND     SM401  ; 常時OFF
      LD      D54.E  ; 異常予備
      ANI     M9  ; アラームリセット中
      ORB
      ANB
      OUT     T178 K0  ; 異常予備  遅延
      AND     T178  ; 異常予備  遅延
      OUT     D54.E  ; 異常予備
1087  LD      SM401  ; 常時OFF
      LD      T10  ; 電源入 遅延
      AND     SM401  ; 常時OFF
      LD      D54.F  ; 異常予備
      ANI     M9  ; アラームリセット中
      ORB
      ANB
      OUT     T179 K0  ; 異常予備  遅延
      AND     T179  ; 異常予備  遅延
      OUT     D54.F  ; 異常予備
; [Title] 警報
1101  LDI     SM400  ; 常時ON
      LD      T10  ; 電源入 遅延
      AND=    K1 D423  ; WMSから_入庫 搬入 RFID異常
      LD      D55.0  ; 入庫側 搬入 RFID 不一致
      ANI     M9  ; アラームリセット中
      ORB
      ANB
      OUT     T180 K0  ; 入庫側 搬入 RFID 不一致  遅延
      AND     T180  ; 入庫側 搬入 RFID 不一致  遅延
      OUT     D55.0  ; 入庫側 搬入 RFID 不一致
1116  LDI     SM400  ; 常時ON
      LD      T10  ; 電源入 遅延
      AND=    K1 D424  ; WMSから_入庫 搬出 RFID異常
      LD      D55.1  ; 入庫側 搬出 計画未達
      ANI     M9  ; アラームリセット中
      ORB
      ANB
      OUT     T181 K0  ; 入庫側 搬出 計画未達  遅延
      AND     T181  ; 入庫側 搬出 計画未達  遅延
      OUT     D55.1  ; 入庫側 搬出 計画未達
